// TIA Portal V19 export
TYPE "C501_VAR_TRA_TYPIC"
   STRUCT
      OBS { ExternalAccessible := 'False'; ExternalVisible := 'False'; ExternalWritable := 'False'} : USInt;   // Observeerbaarheid
   END_STRUCT;
END_TYPE
